Fanuc KAREL source: kt00442.KL

-- PROVISIONAL review KL for V940-1; original PC SHA256 2331eaf6e0f2da51bfe556d46a6c9ba2b9c5a3d50e70741c65d3d2e7c82fc768
-- Incomplete behavior may be omitted. Consult companion uncertainty JSON. Do not deploy.
PROGRAM KT00442
%NOLOCKGROUP
VAR
  R1 : REAL
  R2 : REAL
  OUT : BOOLEAN
BEGIN
  -- V9_ZERO_TABLE_METADATA_HINT layout=0001; no indexed target words; source/name/runtime held
  -- UNRESOLVED_PC offsets 5-16; opcodes 2E,23
  -- UNRESOLVED_PC offsets 21-32; opcodes 2E,23
  -- UNRESOLVED_PC offsets 37-48; opcodes 2E,23
  -- UNRESOLVED_PC offsets 53-64; opcodes 2E,23
  -- UNRESOLVED_PC offsets 69-88; opcodes 21,21,72,23
  -- UNRESOLVED_PC offsets 93-97; opcodes 7F
END KT00442
